// TIA Portal V21 export
VAR_GLOBAL   // PLC tag table "GruppoRiempiSendDigitali"
END_VAR
VAR_GLOBAL CONSTANT   // user constants
   K_SegnaleVersoGruppoRiempi_ChiudiCanstop : Int := 1;
END_VAR
